SYSTEM temexdmodricker
  (* Version 1.0, Author, 4DIAC-Consortium *)
  APPLICATION Loop5
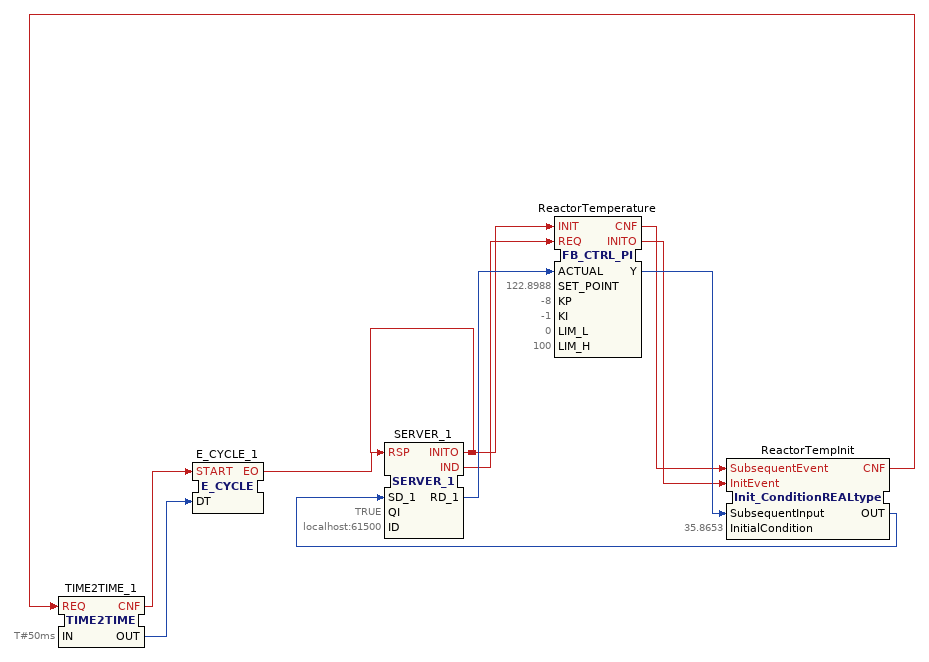
    FBS
      TIME2TIME_1 : TIME2TIME(IN := T#50ms);
      ReactorTemperature : FB_CTRL_PI(SET_POINT := 122.8988, KP := -8, KI := -1, LIM_L := 0, LIM_H := 100);
      ReactorTempInit : Init_ConditionREALtype(InitialCondition := 35.8653);
      E_CYCLE_1 : E_CYCLE;
      SERVER_1 : SERVER_1(QI := TRUE, ID := localhost:61500);
    END_FBS
    EVENT_CONNECTIONS
      ReactorTemperature.CNF TO ReactorTempInit.SubsequentEvent;
      ReactorTemperature.INITO TO ReactorTempInit.InitEvent;
      ReactorTempInit.CNF TO TIME2TIME_1.REQ;
      TIME2TIME_1.CNF TO E_CYCLE_1.START;
      SERVER_1.INITO TO ReactorTemperature.INIT;
      SERVER_1.INITO TO SERVER_1.RSP;
      SERVER_1.IND TO ReactorTemperature.REQ;
      E_CYCLE_1.EO TO SERVER_1.RSP;
    END_CONNECTIONS
    DATA_CONNECTIONS
      ReactorTemperature.Y TO ReactorTempInit.SubsequentInput;
      TIME2TIME_1.OUT TO E_CYCLE_1.DT;
      SERVER_1.RD_1 TO ReactorTemperature.ACTUAL;
      ReactorTempInit.OUT TO SERVER_1.SD_1;
    END_CONNECTIONS
  END_APPLICATION
  DEVICE FORTE_PC : FORTE_PC(MGR_ID := "localhost:61499")
    {SET_ATTRIBUTE(Profile, HOLOBLOC)}
    RESOURCE EMB_RES : EMB_RES
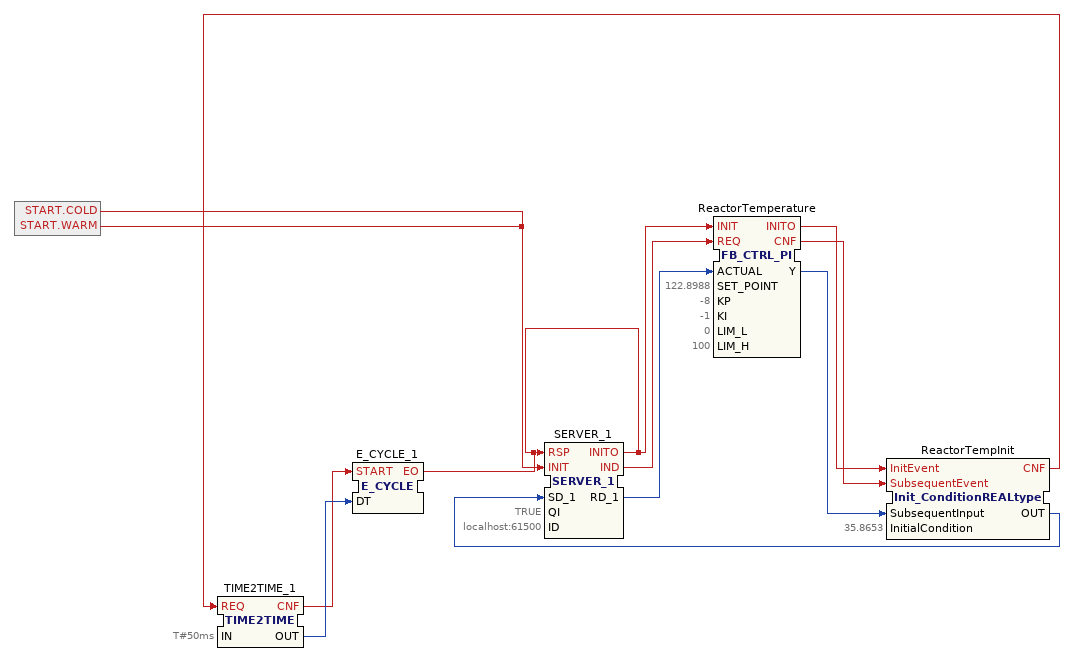
      FBS
        SERVER_1 : SERVER_1(QI := TRUE, ID := localhost:61500);
        TIME2TIME_1 : TIME2TIME(IN := T#50ms);
        ReactorTemperature : FB_CTRL_PI(SET_POINT := 122.8988, KP := -8, KI := -1, LIM_L := 0, LIM_H := 100);
        ReactorTempInit : Init_ConditionREALtype(InitialCondition := 35.8653);
        E_CYCLE_1 : E_CYCLE;
      END_FBS
      EVENT_CONNECTIONS
        SERVER_1.INITO TO SERVER_1.RSP;
        SERVER_1.INITO TO ReactorTemperature.INIT;
        SERVER_1.IND TO ReactorTemperature.REQ;
        ReactorTemperature.INITO TO ReactorTempInit.InitEvent;
        ReactorTemperature.CNF TO ReactorTempInit.SubsequentEvent;
        ReactorTempInit.CNF TO TIME2TIME_1.REQ;
        TIME2TIME_1.CNF TO E_CYCLE_1.START;
        E_CYCLE_1.EO TO SERVER_1.RSP;
        START.COLD TO SERVER_1.INIT;
        START.WARM TO SERVER_1.INIT;
      END_CONNECTIONS
      DATA_CONNECTIONS
        SERVER_1.RD_1 TO ReactorTemperature.ACTUAL;
        ReactorTemperature.Y TO ReactorTempInit.SubsequentInput;
        ReactorTempInit.OUT TO SERVER_1.SD_1;
        TIME2TIME_1.OUT TO E_CYCLE_1.DT;
      END_CONNECTIONS
    END_RESOURCE
  END_DEVICE
  MAPPINGS
    Loop5.TIME2TIME_1 ON FORTE_PC.EMB_RES.TIME2TIME_1;
    Loop5.ReactorTemperature ON FORTE_PC.EMB_RES.ReactorTemperature;
    Loop5.ReactorTempInit ON FORTE_PC.EMB_RES.ReactorTempInit;
    Loop5.E_CYCLE_1 ON FORTE_PC.EMB_RES.E_CYCLE_1;
    Loop5.SERVER_1 ON FORTE_PC.EMB_RES.SERVER_1;
  END_MAPPINGS
  SEGMENTS
    Ethernet : Ethernet;
  END_SEGMENTS
  LINKS
    FORTE_PC => Ethernet;
  END_LINKS
END_SYSTEM
